TYPE EKF_Data : 
	STRUCT
		{attribute 'GUID' := '4651D9AA-F39F-4D87-B1FC-94AB11715483'}
		State : sPosition;
		(*  w1,w2,w3  *)
		wheelSpeed : ARRAY [1..3] OF LREAL;
		P_Start : ARRAY [1..9] OF LREAL;
		timestamp : LREAL;
	END_STRUCT
END_TYPE

(* stored: Version 1.1.0.1, ProductVersion 3.1.4026.13
   DUT EKF_Data: Id {c8bb2a20-8bfb-4d12-be4c-0de955b4692f} *)
